Staubli VAL3: STR_EDIT.pgx

program Str_Edit(string& x_sData, num x_nX, num x_nY)
  local string l_sBuff
  local num l_nKey
  local string l_sOri
begin

  x_nX=min(max(0,x_nX),39)
  x_nY=min(max(0,x_nY),13)
 // x_nLength=min(max(0,x_nLength),39)
  l_sOri=x_sData

  setTextMode(1)
  l_nKey=0
  l_sBuff=x_sData
  while l_nKey!=270 and l_nKey!=255
    gotoxy(x_nX,x_nY)
    setTextMode(0)
    put(left("                              ",nPanelWidthX-x_nX+nPanelLTopX))
    gotoxy(x_nX,x_nY)
    setTextMode(1)
    l_nKey=get(l_sBuff)
    //Enter
    if l_nKey==270
      setTextMode(0)
      x_sData=l_sBuff
    endIf
    //ESC
    if l_nKey==255
      setTextMode(0)
      x_sData= l_sOri
      setTextMode(0)
    endIf
    gotoxy(x_nX,x_nY)
    put(left(l_sBuff+"                    ",nPanelWidthX-x_nX+nPanelLTopX))
    delay(0)
  endWhile
end
